Yaskawa INFORM job: OK_R2_O54(90,90)AWOK.JBI

/JOB
//NAME OK_R2_O54(90,90)AWOK
///FOLDERNAME X4
//POS
///NPOS 74,74,74,4,0,0
///TOOL 0
///POSTYPE PULSE
///PULSE
C00000=93051,-79362,-65205,-778,51067,80227
C00001=125338,4752,11778,-3355,110867,78656
C00002=125338,4752,11778,-3355,110867,78656
C00003=125339,5428,13792,-3329,109979,78685
C00004=125338,4752,11778,-3355,110867,78656
C00005=125193,10566,16887,-3408,110705,78608
C00006=115080,14427,23905,7535,109251,79269
C00007=115024,12462,22117,7526,109345,79255
C00008=115080,14427,23905,7535,109251,79269
C00009=115005,11939,18951,7603,111013,79358
C00010=114782,18324,21018,7636,113026,79408
C00011=113825,18538,21218,7247,113101,79052
C00012=124914,16975,20215,1386,107196,-80319
C00013=124236,11021,16275,1169,106579,-80567
C00014=122697,11964,18588,-2367,106235,-80981
C00015=120670,5046,12163,39,106065,-81841
C00016=120671,5702,14099,39,105210,-81841
C00017=120670,5046,12163,39,106065,-81841
C00018=120669,10918,17333,38,105901,-81841
C00019=120664,13367,22956,36,103700,-81844
C00020=120664,11809,21544,36,103769,-81844
C00021=120664,13367,22956,36,103700,-81844
C00022=122037,10946,17358,470,105896,-81356
C00023=139789,-6887,-4826,-16075,98624,-73872
C00024=138229,-38529,-21283,-19349,54466,-73206
C00025=138229,-40128,-25771,-18928,56305,-73550
C00026=132021,-97421,-62751,309,78611,-78036
C00027=120704,-95876,-65781,23,90169,-81849
C00028=120673,-19519,-17174,19,99492,-81858
C00029=120653,18427,20993,37,117310,-81846
C00030=120655,11367,17955,38,115552,-81845
C00031=121497,-11331,-6525,-860,109222,-81413
C00032=121497,-10892,-5008,-855,108515,-81408
C00033=121497,-11331,-6525,-860,109222,-81413
C00034=120655,11367,17955,38,115552,-81845
C00035=120694,13185,22347,55,113782,-81831
C00036=120694,11662,20968,55,113850,-81831
C00037=120694,13185,22347,55,113782,-81831
C00038=120653,18427,20993,37,117310,-81846
C00039=120651,11571,12338,39,115316,-81848
C00040=120667,-12436,-9975,-5103,110550,80129
C00041=135504,-6240,-6756,-236,112251,85585
C00042=137072,-5922,-4240,285,110866,86165
C00043=120667,-10291,-8310,-5106,110627,80126
C00044=120668,-12803,-11522,-5133,111310,80096
C00045=121608,-8961,-6663,-24134,110298,59927
C00046=120713,-8973,-6672,-24396,110036,59627
C00047=122195,-10499,-10079,-24194,111672,59860
C00048=120668,-12296,-9868,-24722,110258,59302
C00049=120673,-19507,-17125,19,99468,-81858
C00050=120704,-95876,-65781,23,90169,-81849
C00051=130855,-87373,-58995,278,81466,-78422
C00052=131372,-45145,-32571,250,86782,-78233
C00053=120669,-12962,-10380,-28389,117609,-62624
C00054=120672,-9547,-7734,-28423,117721,-62655
C00055=117378,-11156,-8839,-29623,116446,-63749
C00056=120669,-10818,-8721,-28411,117680,-62644
C00057=120669,-13330,-11926,-28606,118283,-62815
C00058=93666,-325,74,-36602,107166,-71202
C00059=77452,19561,17703,-39337,99497,-75563
C00060=123835,-20062,-17823,-35457,109725,-67278
C00061=144992,-23146,-20676,-36805,111374,-65511
C00062=121196,-24675,-20129,-124,101317,-78289
C00063=120667,-12839,-10285,5181,110528,-79304
C00064=117483,-12687,-10169,4149,110720,-81268
C00065=115000,-10818,-8219,3330,110595,-82191
C00066=120668,-13212,-11835,5211,111288,-80066
C00067=120668,-10700,-8629,5184,110608,-80097
C00068=122912,-11017,-9020,24097,109720,-59806
C00069=120670,-9866,-7984,24814,110314,-59255
C00070=117642,-12567,-12784,24203,112644,-59957
C00071=120669,-12924,-10350,24793,110209,-59279
C00072=120669,-12924,-10350,24793,110209,-59279
C00073=-11166,-12924,-10350,24793,47970,-59279
BC00000=116315,528121,247401
BC00001=118548,534731,365992
BC00002=96598,422087,365992
BC00003=96598,422087,365992
BC00004=96598,422087,365992
BC00005=96598,422087,365992
BC00006=96598,422087,365992
BC00007=96599,422087,365990
BC00008=96598,422087,365992
BC00009=96598,422087,365992
BC00010=96598,422087,365992
BC00011=96598,422087,365992
BC00012=185525,429999,383155
BC00013=185525,429999,383155
BC00014=185525,429999,383155
BC00015=185525,429999,383155
BC00016=185525,429999,383155
BC00017=185525,429999,383155
BC00018=185525,429999,383155
BC00019=185525,429999,383155
BC00020=185525,429999,383155
BC00021=185525,429999,383155
BC00022=185525,429999,383155
BC00023=185525,429999,383155
BC00024=149248,429999,383155
BC00025=145045,518566,383155
BC00026=185525,429999,383155
BC00027=335222,413869,348699
BC00028=335222,413869,348699
BC00029=335222,413869,348699
BC00030=335222,413869,348699
BC00031=335222,412333,344398
BC00032=335222,412333,344398
BC00033=335222,412333,344398
BC00034=335222,412333,344398
BC00035=335222,412333,344398
BC00036=335222,412333,344398
BC00037=335222,412333,344398
BC00038=335222,413869,348699
BC00039=335222,413869,348699
BC00040=285982,404347,347521
BC00041=286853,411236,323497
BC00042=286942,411937,321052
BC00043=286943,411937,321058
BC00044=286943,411937,321058
BC00045=333642,414785,288466
BC00046=333642,414785,288466
BC00047=333642,414785,288466
BC00048=327843,408574,309825
BC00049=335222,413869,348699
BC00050=335222,413869,348699
BC00051=131477,429999,359556
BC00052=156375,406403,376234
BC00053=95150,394363,300688
BC00054=95837,399784,281786
BC00055=101774,401952,274222
BC00056=96111,401953,274225
BC00057=96111,401953,274225
BC00058=101774,401952,274222
BC00059=101774,401952,274222
BC00060=154360,402053,274038
BC00061=166630,400995,273888
BC00062=154584,403936,335644
BC00063=146269,404286,347642
BC00064=145567,409698,328731
BC00065=145336,411484,322504
BC00066=145286,411866,321171
BC00067=145286,411866,321171
BC00068=106446,414921,290643
BC00069=105689,413369,294715
BC00070=110263,408915,310247
BC00071=110263,431898,310247
BC00072=110263,523341,310247
BC00073=110263,523341,310247
EC00000=-798156,-740307
EC00001=-798156,-740307
EC00002=-798156,-740307
EC00003=-798156,-740307
EC00004=-798156,-740307
EC00005=-798156,-740307
EC00006=-798156,-740307
EC00007=-798155,-740307
EC00008=-798156,-740307
EC00009=-798156,-740307
EC00010=-798156,-740307
EC00011=-798156,-740307
EC00012=-798156,-740307
EC00013=-798156,-740307
EC00014=-798156,-740307
EC00015=-798156,-740307
EC00016=-798156,-740307
EC00017=-798156,-740307
EC00018=-798156,-740307
EC00019=-798156,-740307
EC00020=-798156,-740307
EC00021=-798156,-740307
EC00022=-798156,-740307
EC00023=-798156,-740307
EC00024=-798156,-740307
EC00025=-798156,-740307
EC00026=-798156,-740307
EC00027=-798156,-740307
EC00028=-798156,-740307
EC00029=-798156,-740307
EC00030=-798156,-740307
EC00031=-798156,-740307
EC00032=-798156,-740307
EC00033=-798156,-740307
EC00034=-798156,-740307
EC00035=-798156,-740307
EC00036=-798156,-740307
EC00037=-798156,-740307
EC00038=-798156,-740307
EC00039=-798156,-740307
EC00040=-798156,-740307
EC00041=-798153,-740306
EC00042=-798153,-740306
EC00043=-798156,-740307
EC00044=-798156,-740307
EC00045=-798156,-740307
EC00046=-798156,-740307
EC00047=-798156,-740307
EC00048=-798156,-740307
EC00049=-798156,-740307
EC00050=-798156,-740307
EC00051=-798156,-740307
EC00052=-798156,-740307
EC00053=-798156,-740307
EC00054=-798156,-740307
EC00055=-798154,-740306
EC00056=-798156,-740307
EC00057=-798156,-740307
EC00058=-798154,-740306
EC00059=-798154,-740306
EC00060=-798155,-740307
EC00061=-798156,-740307
EC00062=-798156,-740307
EC00063=-798156,-740307
EC00064=-798156,-740307
EC00065=-798156,-740307
EC00066=-798156,-740307
EC00067=-798156,-740307
EC00068=-798156,-740307
EC00069=-798156,-740307
EC00070=-798156,-740307
EC00071=-798156,-740307
EC00072=-798156,-740307
EC00073=-798156,-740307
///POSTYPE BASE
///RECTAN
///RCONF 0,0,0,0,1,0,0,0,0,0,0,0,0,0,0,0,0,0,0,0,0,0,0,0
P00006=2.006,1.622,-0.565,0.0000,0.0000,0.0000
P00021=0.073,2.058,-0.109,0.0000,0.0000,0.0000
P00022=2.006,1.622,-0.565,0.0000,0.0000,0.0000
///RCONF 0,0,0,0,0,0,0,0,0,0,0,0,0,0,0,0,0,0,0,0,0,0,0,0
P00023=-2.957,-4.083,2.762,0.0000,0.0000,0.0000
//INST
///DATE 2024/11/19 18:45
///ATTR SC,RW
///GROUP1 RB1,BS1
///GROUP2 ST1
NOP
'OK_r2_O54(90,90)
'Path S1566
SFTOF3D
MOVJ C00000 BC00000 VJ=100.00  +MOVJ EC00000 VJ=100.00
MOVL C00001 BC00001 V=400.0  +MOVJ EC00001 VJ=100.00
SMOVL C00002 BC00002 V=100.0  +MOVJ EC00002
SREFP 3 C00003 BC00003  +REFP EC00003
CALL JOB:SEARCH-R1-S13D
SET P022 P006
SFTON3D P022
SMOVL C00004 BC00004 V=100.0  +MOVJ EC00004
SMOVL C00005 BC00005 V=166.7  +MOVJ EC00005
SMOVL C00006 BC00006 V=100.0  +MOVJ EC00006
SREFP 3 C00007 BC00007  +REFP EC00007
CALL JOB:SEARCH-R1-S13D
SET P022 P006
SFTON3D P022
SMOVL C00008 BC00008 V=100.0  +MOVJ EC00008
SMOVL C00009 BC00009 V=166.7  +MOVJ EC00009
MOVL C00010 BC00010 V=1000.0  +MOVJ EC00010 VJ=100.00
MOVJ C00011 BC00011 VJ=100.00  +MOVJ EC00011 VJ=99.00
'Path S1567
SFTOF3D
MOVJ C00012 BC00012 VJ=100.00  +MOVJ EC00012 VJ=100.00
MOVL C00013 BC00013 V=400.0  +MOVJ EC00013 VJ=100.00
SMOVL C00014 BC00014 V=100.0  +MOVJ EC00014
SMOVL C00015 BC00015 V=50.0  +MOVJ EC00015
SREFP 3 C00016 BC00016  +REFP EC00016
CALL JOB:SEARCH-R1-S13D
SET P023 P006
SFTON3D P023
SMOVL C00017 BC00017 V=60.0  +MOVJ EC00017
SMOVL C00018 BC00018 V=100.0  +MOVJ EC00018
SMOVL C00019 BC00019 V=166.7  +MOVJ EC00019
SREFP 3 C00020 BC00020  +REFP EC00020
CALL JOB:SEARCH-R1-S13D
SET P023 P006
SFTON3D P023
SFTOF3D
SMOVL C00021 BC00021 V=100.0  +MOVJ EC00021
SMOVL C00022 BC00022 V=100.0  +MOVJ EC00022
MOVL C00023 BC00023 V=166.7  +MOVJ EC00023 VJ=100.00
MOVJ C00024 BC00024 VJ=100.00  +MOVJ EC00024 VJ=100.00
MOVJ C00025 BC00025 VJ=100.00  +MOVJ EC00025 VJ=50.00
MOVJ C00026 BC00026 VJ=100.00  +MOVJ EC00026 VJ=100.00
MOVJ C00027 BC00027 VJ=100.00  +MOVJ EC00027 VJ=100.00
MOVJ C00028 BC00028 VJ=15.00  +MOVJ EC00028 VJ=100.00
'Path S1568
SFTOF3D
MOVJ C00029 BC00029 VJ=100.00  +MOVJ EC00029 VJ=100.00
MOVL C00030 BC00030 V=333.3  +MOVJ EC00030 VJ=100.00
SMOVL C00031 BC00031 V=100.0  +MOVJ EC00031
SREFP 3 C00032 BC00032  +REFP EC00032
CALL JOB:SEARCH-R1-S13D
SET P021 P006
SFTON3D P021
SMOVL C00033 BC00033 V=100.0  +MOVJ EC00033
SMOVL C00034 BC00034 V=250.0  +MOVJ EC00034
SMOVL C00035 BC00035 V=100.0  +MOVJ EC00035
SREFP 3 C00036 BC00036  +REFP EC00036
CALL JOB:SEARCH-R1-S13D
SET P021 P006
SFTON3D P021
SMOVL C00037 BC00037 V=100.0  +MOVJ EC00037
MOVL C00038 BC00038 V=1000.0  +MOVJ EC00038 VJ=100.00
MOVJ C00039 BC00039 VJ=100.00  +MOVJ EC00039 VJ=10.00
'Path W1569
SFTOF3D
SFTON3D P021
MOVJ C00040 BC00040 VJ=100.00  +MOVJ EC00040 VJ=100.00
MOVJ C00041 BC00041 VJ=100.00  +MOVJ EC00041 VJ=100.00
SMOVL C00042 BC00042 V=100.0 PL=0  +MOVJ EC00042
SREFP 1 C00043 BC00043  +REFP EC00043
SREFP 2 C00044 BC00044  +REFP EC00044
MACRO1 MJ#(0) ARGF14
ARCON
SMOVL C00045 BC00045 V=10.0  +MOVJ EC00045
SMOVL C00046 BC00046 V=10.0  +MOVJ EC00046
ARCOF
SMOVL C00047 BC00047 V=400.0  +MOVJ EC00047
SMOVL C00048 BC00048 V=1000.0  +MOVJ EC00048
SFTOF3D
MOVJ C00049 BC00049 VJ=100.00  +MOVJ EC00049 VJ=100.00
MOVJ C00050 BC00050 VJ=50.00  +MOVJ EC00050 VJ=100.00
MOVJ C00051 BC00051 VJ=100.00  +MOVJ EC00051 VJ=100.00
MOVJ C00052 BC00052 VJ=25.00  +MOVJ EC00052 VJ=100.00
SFTOF3D
'Path W1570
SFTOF3D
SFTON3D P023
MOVJ C00053 BC00053 VJ=100.00  +MOVJ EC00053 VJ=100.00
SMOVL C00054 BC00054 V=333.3  +MOVJ EC00054
SMOVL C00055 BC00055 V=166.7 PL=0  +MOVJ EC00055
SREFP 1 C00056 BC00056  +REFP EC00056
SREFP 2 C00057 BC00057  +REFP EC00057
MACRO1 MJ#(0) ARGF14
ARCON
SMOVL C00058 BC00058 V=10.0  +MOVJ EC00058
SMOVL C00059 BC00059 V=10.0  +MOVJ EC00059
ARCOF
SMOVL C00060 BC00060 V=400.0  +MOVJ EC00060
SMOVL C00061 BC00061 V=416.7  +MOVJ EC00061
SFTOF3D
MOVJ C00062 BC00062 VJ=100.00  +MOVJ EC00062 VJ=50.00
'Path W1571
SFTOF3D
SFTON3D P022
MOVJ C00063 BC00063 VJ=100.00  +MOVJ EC00063 VJ=100.00
MOVJ C00064 BC00064 VJ=100.00  +MOVJ EC00064 VJ=100.00
SMOVL C00065 BC00065 V=100.0 PL=0  +MOVJ EC00065
SREFP 1 C00066 BC00066  +REFP EC00066
SREFP 2 C00067 BC00067  +REFP EC00067
MACRO1 MJ#(0) ARGF14
ARCON
SMOVL C00068 BC00068 V=10.0  +MOVJ EC00068
ARCOF
SMOVL C00069 BC00069 V=400.0  +MOVJ EC00069
SMOVL C00070 BC00070 V=1000.0  +MOVJ EC00070
SFTOF3D
MOVJ C00071 BC00071 VJ=100.00  +MOVJ EC00071 VJ=100.00
MOVJ C00072 BC00072 VJ=100.00  +MOVJ EC00072 VJ=100.00
MOVJ C00073 BC00073 VJ=70.00  +MOVJ EC00073 VJ=100.00
END
